% RSLogix 500 project Hourmeter.RSS, saved by version 8.40.00.08 %
PROJECT "UNTITLED"    % processor: Bul.1763 MicroLogix 1100 Series B %

PROGRAM FILES
  LAD 2   14 rungs

DATA FILES
  O0 OUTPUT  4 elements
  I1 INPUT  6 elements
  S2 STATUS  66 elements
  B3 BINARY  1 elements
  T4 TIMER  4 elements
  C5 COUNTER  4 elements
  R6 CONTROL  1 elements
  N7 INTEGER  4 elements
  F8 FLOAT  1 elements

LADDER 2
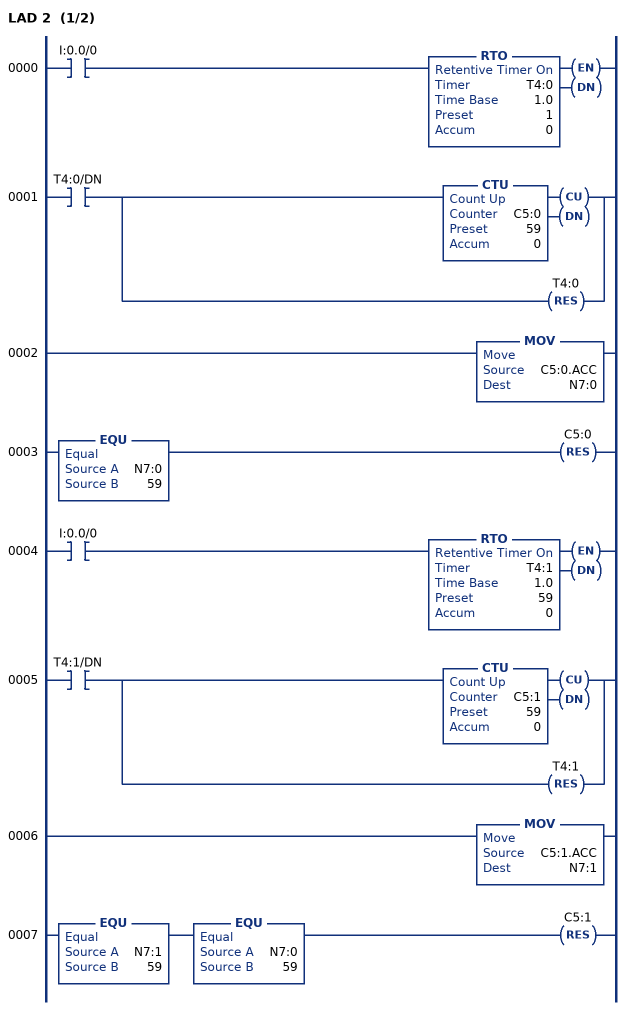
% Rung: 0 %
SOR XIC I:0.0/0 RTO T4:0 1.0 1 0 EOR
% Rung: 1 %
SOR XIC T4:0/DN BST CTU C5:0 59 0 NXB RES T4:0 BND EOR
% Rung: 2 %
SOR MOV C5:0.ACC N7:0 EOR
% Rung: 3 %
SOR EQU N7:0 59 RES C5:0 EOR
% Rung: 4 %
SOR XIC I:0.0/0 RTO T4:1 1.0 59 0 EOR
% Rung: 5 %
SOR XIC T4:1/DN BST CTU C5:1 59 0 NXB RES T4:1 BND EOR
% Rung: 6 %
SOR MOV C5:1.ACC N7:1 EOR
% Rung: 7 %
SOR EQU N7:1 59 EQU N7:0 59 RES C5:1 EOR

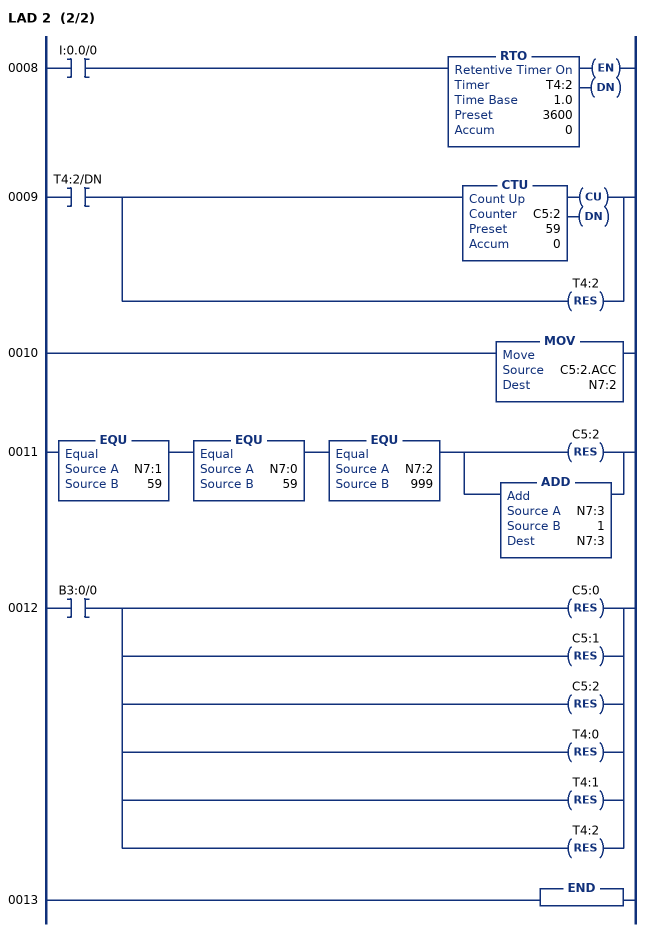
% Rung: 8 %
SOR XIC I:0.0/0 RTO T4:2 1.0 3600 0 EOR
% Rung: 9 %
SOR XIC T4:2/DN BST CTU C5:2 59 0 NXB RES T4:2 BND EOR
% Rung: 10 %
SOR MOV C5:2.ACC N7:2 EOR
% Rung: 11 %
SOR EQU N7:1 59 EQU N7:0 59 EQU N7:2 999 BST RES C5:2 NXB ADD N7:3 1 N7:3 BND EOR
% Rung: 12 %
SOR XIC B3:0/0 BST RES C5:0 NXB RES C5:1 NXB RES C5:2 NXB RES T4:0 NXB RES T4:1 NXB RES T4:2 BND EOR
% Rung: 13 %
SOR END EOR

DATA TABLE (non-zero values as saved)
DATA T4
% .PRE .ACC %
% T4:0 % 1 0
% T4:1 % 59 0
% T4:2 % 3600 0
DATA C5
% .PRE .ACC %
% C5:0 % 59 0
% C5:1 % 59 0
% C5:2 % 59 0
% C5:3 % 59 1
